PROGRAM MAIN
VAR
	(* Messages sent to CCS. *)
	outAxisStatus: AxisStatus;
	outControllerStatus: ControllerStatus;
	outIOStatus: IOStatus;
	ackChangeAxisEnable: ChangeAxisEnable;
	ackChangeOutputLine: ChangeOutputLine;
	ackClearAllFaults: ClearAllFaults;
	ackClearAxisFaults: ClearAxisFaults;
	ackEnableAllAxes: EnableAllAxes;
	ackDisableAllAxes: DisableAllAxes;
	ackMoveAxisRelative: MoveAxisRelative;
	ackMoveAxisAbsolute: MoveAxisAbsolute;
	ackHomeAxis: HomeAxis;
	
	(* Messages coming from CCS. *)
	inChangeAxisEnable: ChangeAxisEnable;
	inChangeOutputLine: ChangeOutputLine;
	inClearAllFaults: ClearAllFaults;
	inClearAxisFaults: ClearAxisFaults;
	inEnableAllAxes: EnableAllAxes;
	inDisableAllAxes: DisableAllAxes;
	inMoveAxisRelative: MoveAxisRelative;
	inMoveAxisAbsolute: MoveAxisAbsolute;
	inHomeAxis: HomeAxis;

	firstCycle: BOOL := TRUE;
END_VAR

VAR CONSTANT
	zeroID: MessageID := (lowUUID := 0, highUUID := 0, dtime := 0, sequence := 0);
END_VAR

(* Initialization. *)
IF firstCycle THEN
	firstCycle := FALSE;
	ackChangeAxisEnable.id := inChangeAxisEnable.id := zeroID;
	ackChangeOutputLine.id := inChangeOutputLine.id := zeroID;
	ackClearAllFaults.id := inClearAllFaults.id := zeroID;
	ackClearAxisFaults.id := inClearAxisFaults.id := zeroID;
	ackEnableAllAxes.id := inEnableAllAxes.id := zeroID;
	ackDisableAllAxes.id := inDisableAllAxes.id := zeroID;
	ackMoveAxisRelative.id := inMoveAxisRelative.id := zeroID;
	ackMoveAxisAbsolute.id := inMoveAxisAbsolute.id := zeroID;
	ackHomeAxis.id := inHomeAxis.id := zeroID;
	
	MSG.changeAxisEnable.CreateEx(TC_EVENTS.CCSEventClass.MsgChangeAxisEnable, 0);
END_IF

(* Check for arrival of new messages. *)
IF haveDifferentIDs(inChangeAxisEnable, ackChangeAxisEnable) THEN
	ackChangeAxisEnable := inChangeAxisEnable;
	printChangeAxisEnable(ackChangeAxisEnable);
END_IF

END_PROGRAM

(* stored: Version 1.1.0.1, ProductVersion 3.1.4022.12
   POU MAIN: Id {4058dd10-e5cd-4d2f-a657-aa9bd7a32e9a}, SpecialFunc None *)
